// TIA Portal V16 export
// export: Created 2021-04-06T19:52:19.3385582Z, ExportSetting WithDefaults, DisplayName Totally Integrated Automation Portal, DisplayVersion V16, DisplayName TIA Portal Version Control Interface, DisplayVersion V16, DisplayName TIA Portal Openness, DisplayVersion V16, DisplayName STEP 7 Professional, DisplayVersion V16, DisplayName STEP 7 Safety, DisplayVersion V16, DisplayName WinCC Unified SCADA Engineering System, DisplayVersion V16
TYPE "plavnik"
// stored: IsFailsafeCompliant false
   STRUCT
      statePlavnik : Bool;   // состояние плавника
      manOpenPlavnik : Bool;   // ручн - открытие клапана
      manClosePlavnik : Bool;   // ручн - закрытие клапана
   END_STRUCT;
END_TYPE
